(*
SPDX-FileCopyrightText: © 2026 Oleksandr Tiutyk <trofimich@gmail.com>
SPDX-License-Identifier: MIT
License: https://opensource.org/license/mit
*)

(*!
<summary>Removes an empty filesystem directory through cyclic task execution.</summary>
<description>
Configure DirectoryPath, PathType, AmsNetId and Timeout before Start and keep them unchanged until STOPPED.
The path must be nonblank and pass PathHelper's limited lexical filter; native services determine whether the
requested operation is supported. This task does not perform an existence precheck or suppress native errors.
Invalid configuration and native errors use the base Task failure and cleanup path. Cancellation waits for
submitted I/O without rolling back completed filesystem changes. Reset clears the native request state and
preserves configuration. Use one owner task per instance.
</description>
*)

{attribute 'no_explicit_call' := 'do not call this function block directly'}
FUNCTION_BLOCK RemoveEmptyDirectory EXTENDS TOF_Tasks.Task IMPLEMENTS IFileSystemTask
VAR_STAT
	//! <summary>Static type metadata available before the base task initializes its default name.</summary>
	{attribute 'hide'}
	_ClassName : STRING := __POUNAME();
END_VAR
VAR
    _RemoveDirectory : Tc2_System.FB_RemoveDir;	
END_VAR

(*!
<summary>Selects the ADS target for the native filesystem operation.</summary>
<description>
Configure before Start and keep unchanged until STOPPED; the setter stores configuration without submitting
I/O.
</description>
*)
{attribute 'monitoring' := 'call'}
PROPERTY AmsNetId : Tc2_System.T_AmsNetID
GET
AmsNetId := _RemoveDirectory.sNetId;
END_GET
SET
_RemoveDirectory.sNetId := AmsNetId;
END_SET
END_PROPERTY

(*!
<summary>Provides the concrete type name used in diagnostics.</summary>
<description>
Returns borrowed read-only metadata; keep the instance alive and do not modify the referenced string.
Initialized static storage is ready during base Task.FB_init; this getter has no side effects or exceptions.
</description>
*)
{attribute 'monitoring' := 'call'}
PROPERTY ClassName : REFERENCE TO STRING
GET
ClassName REF= _ClassName;
END_GET
END_PROPERTY

{attribute 'monitoring' := 'call'}
(*!
<summary>Provides the copied path for the next directory operation.</summary>
<description>
Set before Start and keep unchanged until STOPPED. Checked by PathHelper before submission, then interpreted
by the native service using PathType. Assignment does not perform I/O; Reset preserves it.
</description>
*)
PROPERTY DirectoryPath : Tc2_System.T_MaxString
GET
DirectoryPath := _RemoveDirectory.sPathName;
END_GET
SET
_RemoveDirectory.sPathName := DirectoryPath;
END_SET
END_PROPERTY

(*!
<summary>Provides the library namespace used in diagnostics.</summary>
<description>Returns borrowed read-only namespace storage; do not modify the referenced string.</description>
*)
{attribute 'monitoring' := 'call'}
PROPERTY NamespaceName : REFERENCE TO STRING
GET
NamespaceName REF= CurrentNamespace.Name;
END_GET
END_PROPERTY

(*!
<summary>Resets the native request edge after the task has stopped.</summary>
<description>
Preserves configured inputs and does not undo completed filesystem effects. Pending I/O must finish during
stopping before this hook runs.
</description>
*)
METHOD PROTECTED OnReset
_RemoveDirectory(bExecute := FALSE);
END_METHOD

(*!
<summary>Validates the configured path and advances the native empty-directory removal request.</summary>
<description>
Computed diagnostic strings are held in local buffers for the duration of the receiving call without dynamic
string-builder allocations.
</description>
*)
METHOD PROTECTED OnRunning
VAR_OUTPUT
	processingState : TOF_Tasks.TASK_PROCESSING_STATE;
END_VAR
VAR_IN_OUT
	stopReasonMessage : TOF_Core.ERROR_MESSAGE;
END_VAR
VAR	
	pathErrorMessage : WSTRING(255);
	formattedExceptionMessage : TOF_Core.ERROR_MESSAGE;
END_VAR
IF NOT _RemoveDirectory.bExecute THEN 
	IF TOF_Core.Strings.IsNullOrWhiteSpace(stringToCheck := _RemoveDirectory.sPathName) THEN
		TOF_Core.Exceptions.ThrowDataMemberNotSpecified(
			sourceNamespaceName := NamespaceName,
			sourceClassName := ClassName,
			sourcePOUName := __POUNAME(),
			sourcePosition := __POSITION(),
			dataMemberName := 'DirectoryPath'
		);		
	END_IF
	
	IF NOT PathHelper.IsValidDirectoryPath(directoryPath := _RemoveDirectory.sPathName, errorMessage => pathErrorMessage) THEN
		FileSystemExceptions.ThrowInvalidPath(
			sourceNamespaceName := NamespaceName,
			sourceClassName := ClassName,
			sourcePOUName := __POUNAME(),
			sourcePosition := __POSITION(),
			path := _RemoveDirectory.sPathName,
			errorMessage := pathErrorMessage
		);
	END_IF
END_IF

_RemoveDirectory(bExecute := TRUE);

IF _RemoveDirectory.bError THEN
	TOF_Core.WideStrings.Append255(
		formattedExceptionMessage,
		"An while removing directory '",
		TO_WSTRING(_RemoveDirectory.sPathName),
		"'");

	FileSystemExceptions.ThrowFileSystem(
		sourceNamespaceName := NamespaceName,
		sourceClassName := ClassName,
		sourcePOUName := __POUNAME(),
		sourcePosition := __POSITION(),
		message := formattedExceptionMessage,
		errorCode := _RemoveDirectory.nErrId
	);
END_IF

IF NOT _RemoveDirectory.bBusy THEN
	processingState := TOF_Tasks.TASK_PROCESSING_STATE.DONE;
END_IF
END_METHOD

(*!
<summary>Waits for an already submitted operation before task termination.</summary>
<description>
Runs for every stop reason. Advances the pending FB with bExecute=FALSE without issuing another request.
Completion does not roll back side effects. Keep configuration and borrowed buffers valid until STOPPED.
</description>
<param name="readyToRelease">TRUE when the underlying FB is no longer busy.</param>
*)
METHOD PROTECTED OnStopping
VAR_OUTPUT
	readyToRelease : BOOL;
END_VAR
IF _RemoveDirectory.bBusy THEN
	_RemoveDirectory(bExecute := FALSE);
END_IF

readyToRelease := NOT _RemoveDirectory.bBusy;
END_METHOD

(*!
<summary>Selects the native path context for the filesystem request.</summary>
<description>
Configure before Start and keep unchanged until STOPPED. It is passed to the native operation, not used as a
path-validity result. Reset preserves it.
</description>
*)
{attribute 'monitoring' := 'call'}
PROPERTY PathType : Tc2_System.E_OpenPath
GET
PathType := _RemoveDirectory.ePath;
END_GET
SET
_RemoveDirectory.ePath := PathType;
END_SET
END_PROPERTY

(*!
<summary>Reports the size of this concrete instance in bytes.</summary>
*)
{attribute 'monitoring' := 'call'}
PROPERTY SelfSize : ULINT
GET
SelfSize := XSIZEOF(THIS^);
END_GET
END_PROPERTY

(*!
<summary>Configures the timeout passed to native operation requests.</summary>
<description>
Set before Start and keep unchanged until STOPPED. Reset preserves this value. It is not an overall task
deadline or a guarantee of resource release after a timeout.
</description>
*)
{attribute 'monitoring' := 'call'}
PROPERTY Timeout : TIME
GET
Timeout := _RemoveDirectory.tTimeout;
END_GET
SET
_RemoveDirectory.tTimeout := Timeout;
END_SET
END_PROPERTY

END_FUNCTION_BLOCK

(* stored: Version 1.1.0.1
   POU RemoveEmptyDirectory: Id {f7699339-eb16-4c49-8ff9-e8b510a181bf}, SpecialFunc None
   Folder Inputs: Id {3c1b2bb2-508a-43ab-aba6-d51610d36987}
   Folder Members to override: Id {80e81cc0-48cb-4c8d-a6d2-f5019c2649ac}
   Property AmsNetId: Id {e619447a-91f5-4cfd-87c1-c6f4d65469a7}
   Get Get: Id {af838fb5-84a9-40c2-96ed-bb37e1ba8ee8}
   Set Set: Id {955f8a77-cfbb-437a-a3ea-c4c2072c8db2}
   Property ClassName: Id {9bdfd013-5a24-4a24-9847-b8d276cbdfd1}
   Get Get: Id {07f43309-f5f9-4714-8a79-b20e37081f91}
   Property DirectoryPath: Id {d94128c9-a1f4-40bf-a870-d7916c828353}
   Get Get: Id {1f72f3d7-a990-4668-a6c3-c54f2f298ded}
   Set Set: Id {39cb2b34-0284-49a9-954b-190ef76241ef}
   Property NamespaceName: Id {c30ceec4-6b12-4987-9c9a-253d7cedcfe2}
   Get Get: Id {5de19f01-2439-4806-bb38-5c646f83ed28}
   Method OnReset: Id {054f9fa5-a632-419e-a47f-3fd2edb96643}
   Method OnRunning: Id {df915afb-aa65-445f-a579-78975326fa79}
   Method OnStopping: Id {d399643c-23a2-4f0b-a5c6-299e72a07996}
   Property PathType: Id {2b9d54ab-fa46-41da-ac42-cdc7d5acef43}
   Get Get: Id {6baf4074-7f57-4b46-a346-9359d4fc170d}
   Set Set: Id {7a03c98f-e798-4494-b934-37bb17268ced}
   Property SelfSize: Id {9adbdd4e-26f1-45e1-9314-6ac5a9fcf883}
   Get Get: Id {7af252a4-6350-4943-9c1e-b0b9f893fccd}
   Property Timeout: Id {c5f42126-d467-415e-a93a-fa9d11d77a43}
   Get Get: Id {3464bdc4-4947-406d-8d6a-94c7e64bc5b4}
   Set Set: Id {67cf6448-3dc3-4665-a07b-57b154ad6605} *)
